// TIA Portal V16 export
// export: Created 2023-03-29T11:04:42.5920497Z, ExportSetting WithDefaults, DisplayName Totally Integrated Automation Portal, DisplayVersion V16 Update 6, DisplayName TIA Portal Version Control Interface, DisplayVersion V16 Update 2, DisplayName TIA Portal Openness, DisplayVersion V16 Update 6, DisplayName STEP 7 Professional, DisplayVersion V16 Update 6, DisplayName STEP 7 Safety, DisplayVersion V16, DisplayName WinCC Advanced, DisplayVersion V16 Update 6
DATA_BLOCK "temp_dbHoldRegSlave_to_MT101"   // DB102
{ S7_Optimized_Access := 'FALSE' }
VERSION : 0.1
// stored: AutoNumber false, DBAccessibleFromOPCUA true, IsOnlyStoredInLoadMemory false, IsWriteProtectedInAS false
   VAR
      Status_Sterowanie : Struct
         instPump1 : Int;   // Pompa Status M1
         instPump2 : Int := 0;   // Pompa Status M2
         instPump3 : Int := 0;   // Pompa Status M3
         instPump4 : Int := 0;   // Pompa Status M4
         instvValveZ1 : Int := 0;   // Zasuwa Status Z1
         instvValveZ2 : Int := 0;   // Zasuwa Status Z2
         instvValveZ3 : Int := 0;   // Zasuwa Status Z3
         instvValveZ4 : Int := 0;   // Zasuwa Status Z4
         instvValveZ5 : Int := 0;   // Zasuwa Status Z5
         instvValveZ6 : Int := 0;   // Zasuwa Status Z6
         instvValveZ7 : Int := 0;   // Zasuwa Status Z7
         instvValveZ8 : Int := 0;   // Zasuwa Status Z8
         instvValveZ9 : Int := 0;   // Zasuwa Status Z9
         instvValveZ10 : Int := 0;   // Zasuwa Status Z10
         instvValveZ11 : Int := 0;   // Zasuwa Status Z11
         instvValveZ12 : Int := 0;   // Zasuwa Status Z12
         instControllDrivers_1 : Int := 0;   // Bity sterowania napędami (start, stop, otwórz, zamknij) / Bity sterowania napędami (start, stop, otwórz, zamknij) Pompami M1-M4, Zasuwami Z1, Z2, Z3, Z4
         instControllDrivers_2 : Int := 0;   // Bity przełączenia trybu pracy napędów / Bity sterowania napędami ( otwórz, zamknij, start, stop) Zasuwami Z5, Z6, Z7, Z8, Z9, Z10, Z11, Z12
         instConrol_ManAut_1 : Int := 0;   // Bity przełączenia trybu pracy napędów / Bity przełączenia trybu pracy napędów M1-M4, Zasuwami Z1, Z2, Z3, Z4
         instConrol_ManAut_2 : Int := 0;   // Bity przełączenia trybu pracy napędów / Bity przełączenia trybu pracy napędów Z5, Z6, Z7, Z8, Z9, Z10, Z11, Z12
         instLevelTank1 : Int := 0;   // Poziom zbiornik
         instLevelTank2 : Int := 0;   // Poziom zbiornik
         instLevelTank3 : Int := 0;   // Poziom zbiornik
         instLevelTank4 : Int := 0;   // Poziom zbiornik
         instPosition_Z10 : Int := 0;   // rezerwa / Zadawanie położenia Z10
         instControlClearFault1 : Int := 0;   // Bity kasowania alarmów napędów M1-M4, Z1 - Z12
         instControlSygSter_1 : Int := 0;   // rezerwa / Sygnały sterowania strategią (Bit 53.0 - Wyłączony), (Bit 53.1 - Dosilanie), (Bit 53.2 - Przetłączanie), (Bit 53.3 - Automat), (Bit 53.4 - Ręczne )
         instControlSygSter_2 : Int := 0;   // Sygnały sterowania cyklem (Bit 55.0 - Cykl wyłączony (Bit 55.1 - Cykl dobowy), (Bit 55.2 - Cykl tygodniowy), (Bit 55.3 - Cykl ręczny)
         instCurrent_Inverter : Int := 0;   // Aktualny prądu falownika
         instHz_Inverter : Int := 0;   // Aktualne Hz na falowniku
      END_STRUCT;
      Pomiary : Struct
         instLevelSetfilling : Real;   // Zadany poziom napełniania
         instLevelSetemptying : Real;   // Zadany poziom opróżniania
         instSetbarDN500_B6 : Real;   // Zadany ciśnienie tłóczenia kierunek miasto, Modbus 40035
         instSetbarDN500_B5 : Real;   // Zadana ciśnienie dosilania kierunek dosilanie "0" Modbus 40037
         instSetBarMinB9 : Real;   // Zadawana dolna granica ciśnienia studnia "Granica" Modbus 40039
         instB5bar_act : Real;   // Aktualne ciśnienie zasilania z sieci
         instB6bar_act : Real;   // Aktualne ciśnienie DN225 tłoczny
         instB7bar_act : Real;   // Aktualne ciśnienie DN225 pompy
         instB8bar_act : Real;   // Aktualne ciśnienie ssoncy pomp (zab. Suchobieg)
         instPozitionZ10_act : Real;   // Aktualna pozycja zasuwy Z10
         instFlowDN225_act : Real;   // Przepływ DN225 aktualny MIASTO
         instFlowDN225_sum : Real;   // SUMA przepływu Dolna DN225
         instFlowDN500_act : Real;   // Przepływ DN500 (l/s) aktualny, zasilanie zbiorników, DOSILANIE, Modbus 40055
         instFlowDN500_sum : Real;   // SUMA przepływu Dolna DN500 Modbus 40057
      END_STRUCT;
      Godziny : Struct
         instHourStart_Filling : Int;   // Godzina start napełniania
         instMinutStart_Filling : Int;   // Minuta start napełniania
         instHourStop_Filling : Int;   // Godzina stop napełniania
         instMinutStopt_Filling : Int;   // Minuta stop napełniania
         instHourStart_City : Int;   // Godzina start przetłaczanie miasto DN225
         instMinutStart_City : Int;   // Minuty start przetłaczanie miasto DN225
         instHourStop_City : Int;   // Godzina stop przetłaczanie miasto DN225
         instMinutStopt_City : Int;   // Minuty stop przetłaczanie miasto DN225
         instHourStart_Replen : Int;   // Godzina start przetłaczanie miasto DN225
         instMinutStart_Replen : Int;   // Minuty start przetłaczanie miasto DN225
         instHourStop_Replen : Int;   // Godzina stop przetłaczanie miasto DN225
         instMinutStopt_Replen : Int;   // Minuty stop przetłaczanie miasto DN225
      END_STRUCT;
   END_VAR
BEGIN
END_DATA_BLOCK
